// TIA Portal V16 export
// export: Created 2021-07-12T14:47:15.7802802Z, ExportSetting WithDefaults, DisplayName Totally Integrated Automation Portal, DisplayVersion V16, DisplayName TIA Portal Version Control Interface, DisplayVersion V16, DisplayName TIA Portal Openness, DisplayVersion V16, DisplayName STEP 7 Professional, DisplayVersion V16, DisplayName STEP 7 Safety, DisplayVersion V16, DisplayName WinCC Professional, DisplayVersion V16
DATA_BLOCK "HydAxisAnalog2_Data"   // DB33131
{ S7_Optimized_Access := 'TRUE' }
FAMILY : SimaHydTO
VERSION : 1.0
// stored: AutoNumber true, DBAccessibleFromOPCUA true, InstanceOfName LSimaHydTO_typeAxisData, InstanceOfType UDT, IsOnlyStoredInLoadMemory false, IsWriteProtectedInAS false
"LSimaHydTO_typeAxisData"
   // VAR
   //    Velocity : LReal;
   //    Acceleration : LReal;
   //    Position : LReal;
   //    Force : LReal;
   //    ActualVelocity : LReal;
   //    ActualSpeed : LReal;
   //    ActualAcceleration : LReal;
   //    ActualPosition : LReal;
   //    ActualForce : LReal;
   //    Actor { S7_SetPoint := 'True'} : "LSimaHydTO_typeActor";
   //    ValveCharacteristic { S7_SetPoint := 'True'} : "LSimaHydTO_typeValveCharacteristic";
   //    ForceLimits { S7_SetPoint := 'True'} : "LSimaHydTO_typeForceLimits";
   //    Pressure_A_Transducer { S7_SetPoint := 'True'} : "LSimaHydTO_typeTransducer";
   //    Pressure_B_Transducer { S7_SetPoint := 'True'} : "LSimaHydTO_typeTransducer";
   //    PositionControl { S7_SetPoint := 'True'} : "LSimaHydTO_typePositionControl";
   //    ForceControl { S7_SetPoint := 'True'} : "LSimaHydTO_typeForceControl";
   //    DynamicAxisModel { S7_SetPoint := 'True'} : "LSimaHydTO_typeDynamicAxisModel";
   //    SmoothingFilter { S7_SetPoint := 'True'} : "LSimaHydTO_typeSmoothingFilter";
   //    StatusActor { S7_SetPoint := 'True'} : "LSimaHydTO_typeStatusActor";
   //    StatusVChar { S7_SetPoint := 'True'} : "LSimaHydTO_typeStatusVChar";
   //    Status_A_Transducer { S7_SetPoint := 'True'} : "LSimaHydTO_typeStatusTransducer";
   //    Status_B_Transducer { S7_SetPoint := 'True'} : "LSimaHydTO_typeStatusTransducer";
   //    StatusServo { S7_SetPoint := 'True'} : "LSimaHydTO_typeStatusServo";
   //    StatusForce { S7_SetPoint := 'True'} : "LSimaHydTO_typeStatusForce";
   //    StatusForceProfile { S7_SetPoint := 'True'} : "LSimaHydTO_typeStatusForceProfile";
   //    ErrorWord : DWord;
   //    ErrorDetail { S7_SetPoint := 'True'} : "LSimaHydTO_typeErrorDetail";
   //    "Name" { S7_SetPoint := 'True'} : WString[24] := WSTRING#'ANALOG 2';
   //    TO_Axis : DB_ANY;
   //    DataInitialized : Bool;
   //    Internal { S7_SetPoint := 'True'} : "LSimaHydTO_typeInternal";
   // END_VAR
BEGIN
   ValveCharacteristic.DB_NUMBER := 33141;
END_DATA_BLOCK
